INTERFACE I_Scale EXTENDS I_ComponentBase

METHOD Tare
VAR_INPUT
END_VAR
END_METHOD

PROPERTY Weight : LREAL
GET
END_GET
SET
END_SET
END_PROPERTY

END_INTERFACE

(* stored: Version 1.1.0.1
   Itf I_Scale: Id {de0ee560-1e0d-444d-b634-c8840355f512}
   Method Tare: Id {fefcbd18-ee4a-4b17-b26b-df8fcd989e3f}
   Property Weight: Id {cba467ec-8158-4207-8c07-1c9895c7e902}
   Get Get: Id {7d66297f-b009-4e67-87dd-187675222ea3}
   Set Set: Id {ee9c65e6-2f59-4a16-82c3-35f67a947dec} *)
